FUNCTION_BLOCK ResetDetect (* Composite Function Block Type *)
  (* Standard: 61499-2 *)
  (* Version 0.0, 7/28/2023, vv263, nxtControl GmBH, template *)
  PACKAGE Main;
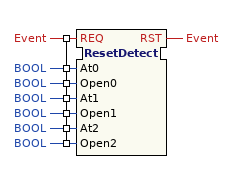
  EVENT_INPUT
    REQ WITH At0, Open0, At1, Open1, At2, Open2; (* Normal Execution Request *)
  END_EVENT
  EVENT_OUTPUT
    RST; (* Execution Confirmation *)
  END_EVENT
  VAR_INPUT
    At0 : BOOL; (* Input event qualifier *)
    Open0 : BOOL;
    At1 : BOOL;
    Open1 : BOOL;
    At2 : BOOL;
    Open2 : BOOL;
  END_VAR
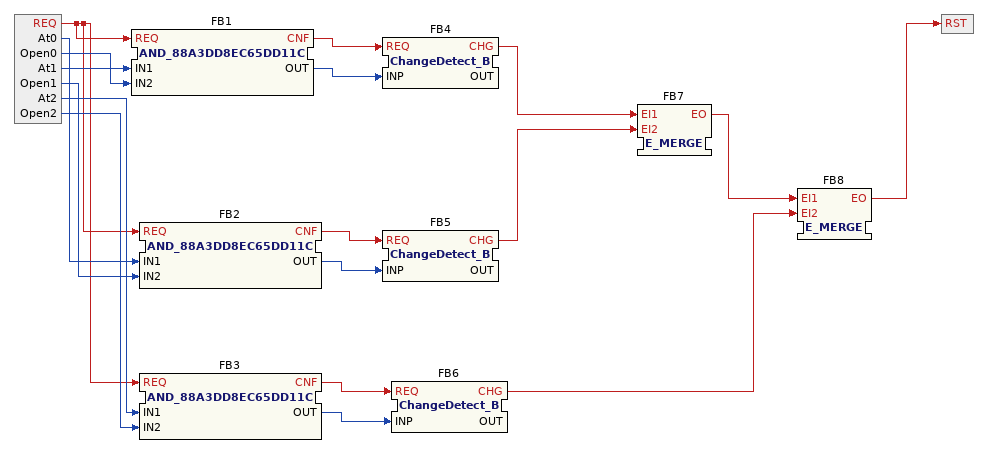
  FBS
    FB1 : AND_88A3DD8EC65DD11C; {SET_ATTRIBUTE(Configuration.GenericFBType.InterfaceParams, Runtime.Standard#CNT:=2;OUT:BOOL)}
    FB2 : AND_88A3DD8EC65DD11C; {SET_ATTRIBUTE(Configuration.GenericFBType.InterfaceParams, Runtime.Standard#CNT:=2;OUT:BOOL)}
    FB3 : AND_88A3DD8EC65DD11C; {SET_ATTRIBUTE(Configuration.GenericFBType.InterfaceParams, Runtime.Standard#CNT:=2;OUT:BOOL)}
    FB4 : ChangeDetect_B;
    FB5 : ChangeDetect_B;
    FB6 : ChangeDetect_B;
    FB7 : E_MERGE;
    FB8 : E_MERGE;
  END_FBS
  EVENT_CONNECTIONS
    REQ TO FB1.REQ;
    REQ TO FB2.REQ;
    REQ TO FB3.REQ;
    FB1.CNF TO FB4.REQ;
    FB2.CNF TO FB5.REQ;
    FB3.CNF TO FB6.REQ;
    FB7.EO TO FB8.EI1;
    FB6.CHG TO FB8.EI2;
    FB4.CHG TO FB7.EI1;
    FB5.CHG TO FB7.EI2;
    FB8.EO TO RST;
  END_CONNECTIONS
  DATA_CONNECTIONS
    At0 TO FB1.IN1;
    Open0 TO FB1.IN2;
    FB1.OUT TO FB4.INP;
    At1 TO FB2.IN1;
    Open1 TO FB2.IN2;
    FB2.OUT TO FB5.INP;
    At2 TO FB3.IN1;
    Open2 TO FB3.IN2;
    FB3.OUT TO FB6.INP;
  END_CONNECTIONS
END_FUNCTION_BLOCK
